Universal Robots PolyScope program: Project1pick2.urp

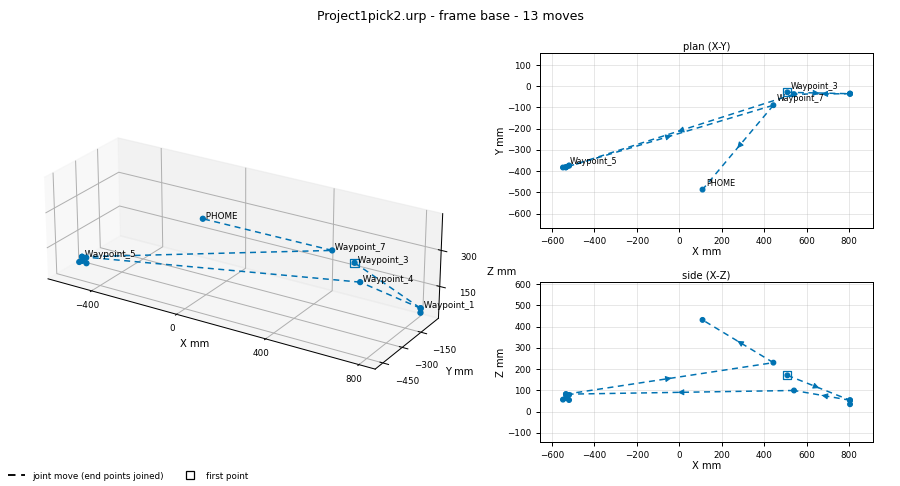
[picture p0: tool path of Project1pick2.urp in frame base, 13 of 13 moves have a stored position in this frame; points joined in program order, loops and branches not executed]
Program Project1pick2 (installation=admin directory=/programs/TUES_530PM createdIn=3.15.8.106339 lastSavedIn=3.15.8.106339 robotSerialNumber=2015350926)
Calibrated DH parameters: a=[0, -0.425, -0.39225, 0, 0, 0]; d=[0.089159, 0, 0, 0.10915, 0.09465, 0.0823]; alpha=[1.570796, 0, 0, 1.570796, -1.570796, 0]; deltaTheta=[0, 0, 0, 0, 0, 0]
Robot Program (runOnlyOnce=true)
  Set DigitalOutput pin=digital_out[0]; digitalValue=0
  Set DigitalOutput pin=digital_out[1]; digitalValue=0
  MoveJ speed 60 deg/s, acceleration 80 deg/s^2 (useActiveTCP=true)
    Waypoint Waypoint_3: TCP in base x=508.862 y=-28.636 z=170.727 mm, rx=-2.197 ry=-2.2407 rz=-0.0052 rad; joints [-195.631, -76.368, 115.777, -129.324, -89.737, -196.76] deg
    Waypoint Waypoint_1: TCP in base x=804.112 y=-35.22 z=53.434 mm, rx=2.1996 ry=-2.2382 rz=0.0055 rad; joints [-190.273, -32.939, 61.013, -118.124, -90.28, -9.278] deg
    Waypoint Waypoint_2: TCP in base x=804.119 y=-35.218 z=34.566 mm, rx=2.1997 ry=-2.2382 rz=0.0057 rad; joints [-190.273, -31.534, 61.288, -119.812, -90.278, -9.278] deg
    Wait Sleep waitTime=0.5
    Set DigitalOutput pin=digital_out[0]; digitalValue=1
    Wait Sleep waitTime=0.5
    Waypoint Waypoint_1: TCP in base x=804.112 y=-35.22 z=53.434 mm, rx=2.1996 ry=-2.2382 rz=0.0055 rad; joints [-190.273, -32.939, 61.013, -118.124, -90.28, -9.278] deg
    Waypoint Waypoint_4: TCP in base x=540.198 y=-37.26 z=99.373 mm, rx=2.1998 ry=-2.2382 rz=0.0056 rad; joints [-195.533, -65.483, 114.099, -138.697, -90.269, -14.542] deg
    Waypoint Waypoint_5: TCP in base x=-534.595 y=-381.84 z=81.964 mm, rx=0.0179 ry=3.1368 rz=0.0001 rad; joints [-334.042, -52.242, 93.855, -131.367, -89.88, -63.39] deg
    Waypoint Waypoint_6: TCP in base x=-548.456 y=-382.853 z=56.301 mm, rx=0.018 ry=3.1369 rz=0.0001 rad; joints [-334.489, -48.699, 92.085, -133.146, -89.886, -63.832] deg
    Wait Sleep waitTime=0.5
    Set DigitalOutput pin=digital_out[0]; digitalValue=0
    Wait Sleep waitTime=0.5
    Waypoint Waypoint_8: TCP in base x=-534.54 y=-381.876 z=64.01 mm, rx=0.0177 ry=3.1367 rz=0.0001 rad; joints [-334.037, -50.6, 94.27, -133.42, -89.879, -63.39] deg
    Wait Sleep waitTime=0.5
    Set DigitalOutput pin=digital_out[0]; digitalValue=1
    Loop While (checkContinuously=false) expression=force()≤50
      Waypoint Waypoint_9: TCP in base x=-519.781 y=-373.985 z=54.328 mm, rx=0.0194 ry=3.137 rz=-0.0012 rad; joints [-334.099, -51.286, 97.631, -136.134, -89.845, -63.39] deg
    Wait Sleep waitTime=0.5
    Set DigitalOutput pin=digital_out[1]; digitalValue=1
    Wait Sleep waitTime=2.5
    Waypoint Waypoint_10: TCP in base x=-519.789 y=-373.981 z=78.734 mm, rx=0.0194 ry=3.1371 rz=-0.0013 rad; joints [-334.1, -53.628, 97.124, -133.288, -89.845, -63.39] deg
    Set DigitalOutput pin=digital_out[0]; digitalValue=0
    Wait Sleep waitTime=0.5
    Waypoint Waypoint_5: TCP in base x=-534.595 y=-381.84 z=81.964 mm, rx=0.0179 ry=3.1368 rz=0.0001 rad; joints [-334.042, -52.242, 93.855, -131.367, -89.88, -63.39] deg
    Waypoint Waypoint_7: TCP in base x=442.98 y=-89.507 z=230.504 mm, rx=-3.1415 ry=0.0179 rz=-0.0077 rad; joints [-205.422, -89.045, 119.992, -121.202, -89.878, -114.771] deg
    Waypoint PHOME: TCP in base x=109.137 y=-486.932 z=431.878 mm, rx=0 ry=3.1414 rz=-0.0004 rad; joints [89.997, -89.999, 90, -90.015, -89.991, -0.004] deg
